TYPE ST_HnltCnLinkageControl :
STRUCT	
	bHeatingMode : BOOL;
	fTargetTemperature_ProductionHall : REAL;
	bAlgorithmPermission_HNLT : BOOL;
	bAlgorithmPermission_CN : BOOL;
	bSetStatusOn_HeatPump : BOOL;
END_STRUCT
END_TYPE

(* stored: Version 1.1.0.1, ProductVersion 3.1.4024.10
   DUT ST_HnltCnLinkageControl: Id {f7c1de2f-a4d7-42fd-89b5-954c364eebb1} *)
